TYPE HydraulicsPumpsGroupIOStatuses :
STRUCT
	///Is the I/O in a healthy state?
	healthStatus: HealthStatus;
END_STRUCT
END_TYPE

(* stored: Version 1.1.0.1, ProductVersion 3.1.4019.2
   DUT HydraulicsPumpsGroupIOStatuses: Id {d959090f-d7ae-48c2-9a13-fcbc05cb75e4} *)
